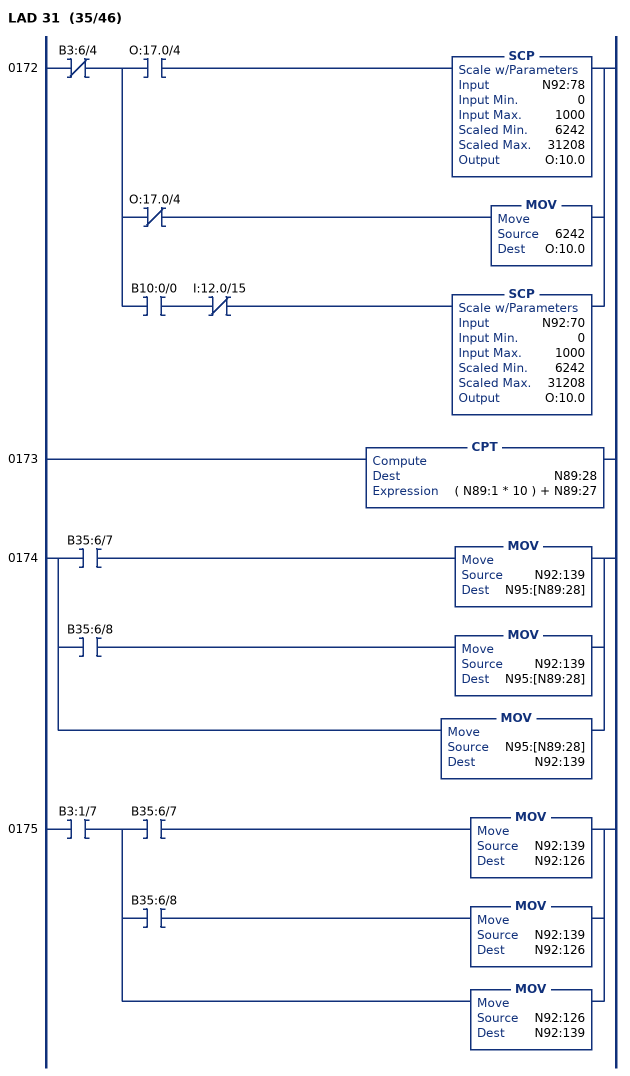
% Rung: 172 %
SOR XIO B3:6/4 BST XIC O:17.0/4 SCP N92:78 0 1000 6242 31208 O:10.0 NXB XIO O:17.0/4 MOV 6242 O:10.0 NXB XIC B10:0/0 XIO I:12.0/15 SCP N92:70 0 1000 6242 31208 O:10.0 BND EOR
% Rung: 173 %
SOR CPT N89:28 " ( N89:1 * 10 ) + N89:27 " EOR
% Rung: 174 %
SOR BST XIC B35:6/7 MOV N92:139 N95:[N89:28] NXB XIC B35:6/8 MOV N92:139 N95:[N89:28] NXB MOV N95:[N89:28] N92:139 BND EOR
% Rung: 175 %
SOR XIC B3:1/7 BST XIC B35:6/7 MOV N92:139 N92:126 NXB XIC B35:6/8 MOV N92:139 N92:126 NXB MOV N92:126 N92:139 BND EOR

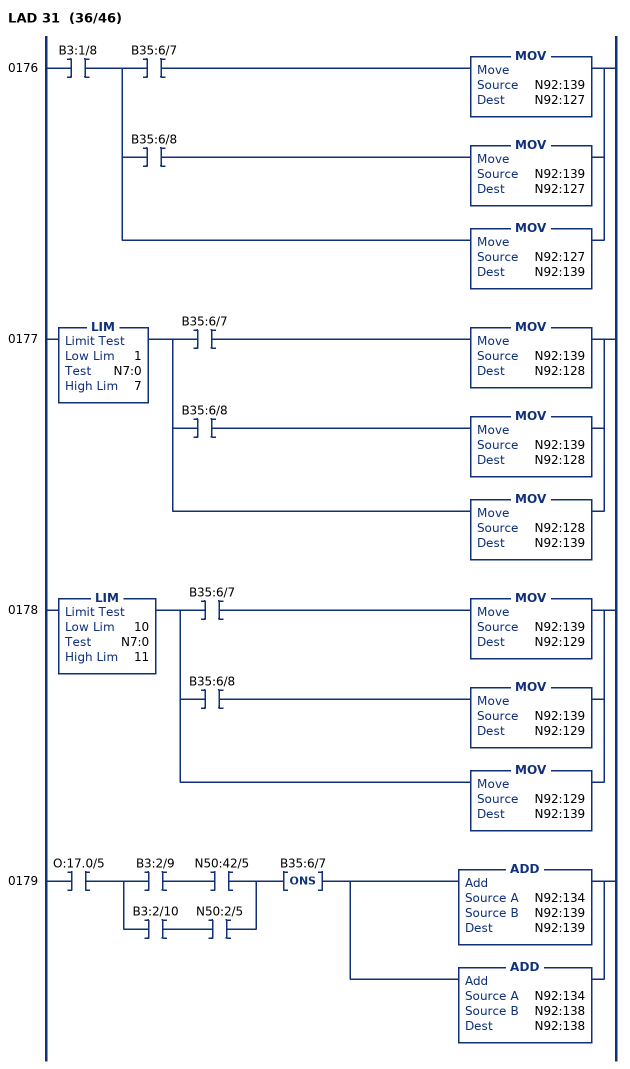
% Rung: 176 %
SOR XIC B3:1/8 BST XIC B35:6/7 MOV N92:139 N92:127 NXB XIC B35:6/8 MOV N92:139 N92:127 NXB MOV N92:127 N92:139 BND EOR
% Rung: 177 %
SOR LIM 1 N7:0 7 BST XIC B35:6/7 MOV N92:139 N92:128 NXB XIC B35:6/8 MOV N92:139 N92:128 NXB MOV N92:128 N92:139 BND EOR
% Rung: 178 %
SOR LIM 10 N7:0 11 BST XIC B35:6/7 MOV N92:139 N92:129 NXB XIC B35:6/8 MOV N92:139 N92:129 NXB MOV N92:129 N92:139 BND EOR
% Rung: 179 %
SOR XIC O:17.0/5 BST XIC B3:2/9 XIC N50:42/5 NXB XIC B3:2/10 XIC N50:2/5 BND OSR B35:6/7 BST ADD N92:134 N92:139 N92:139 NXB ADD N92:134 N92:138 N92:138 BND EOR

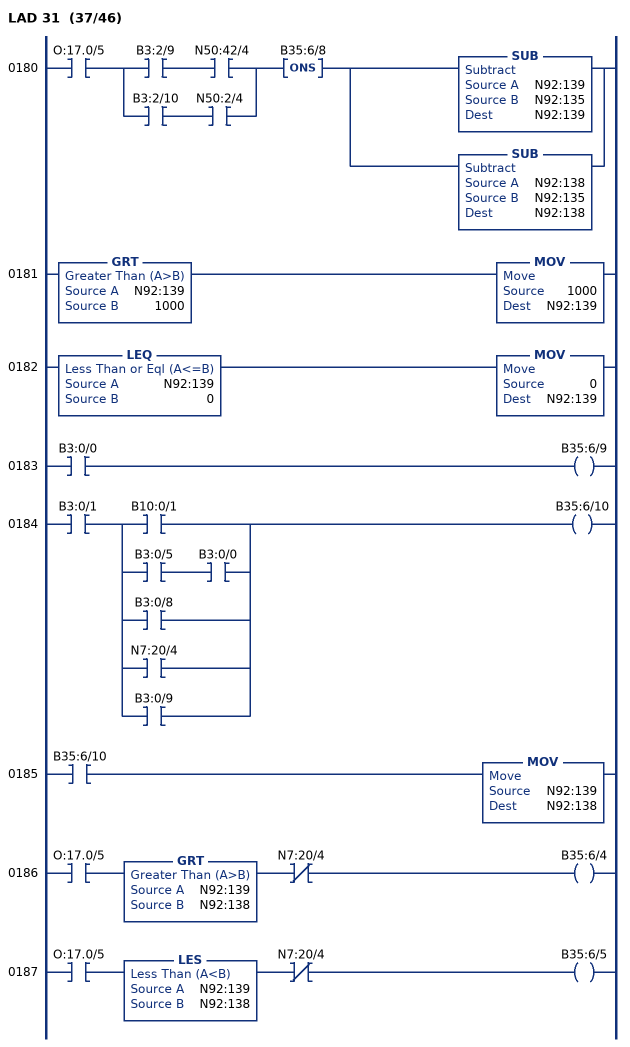
% Rung: 180 %
SOR XIC O:17.0/5 BST XIC B3:2/9 XIC N50:42/4 NXB XIC B3:2/10 XIC N50:2/4 BND OSR B35:6/8 BST SUB N92:139 N92:135 N92:139 NXB SUB N92:138 N92:135 N92:138 BND EOR
% Rung: 181 %
SOR GRT N92:139 1000 MOV 1000 N92:139 EOR
% Rung: 182 %
SOR LEQ N92:139 0 MOV 0 N92:139 EOR
% Rung: 183 %
SOR XIC B3:0/0 OTE B35:6/9 EOR
% Rung: 184 %
SOR XIC B3:0/1 BST XIC B10:0/1 NXB XIC B3:0/5 XIC B3:0/0 NXB XIC B3:0/8 NXB XIC N7:20/4 NXB XIC B3:0/9 BND OTE B35:6/10 EOR
% Rung: 185 %
SOR XIC B35:6/10 MOV N92:139 N92:138 EOR
% Rung: 186 %
SOR XIC O:17.0/5 GRT N92:139 N92:138 XIO N7:20/4 OTE B35:6/4 EOR
% Rung: 187 %
SOR XIC O:17.0/5 LES N92:139 N92:138 XIO N7:20/4 OTE B35:6/5 EOR

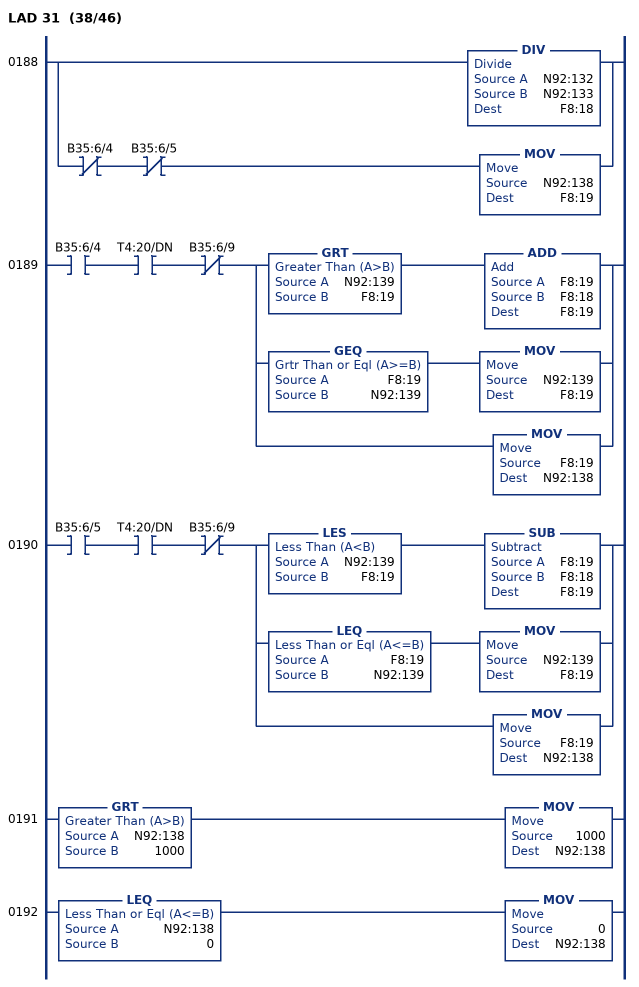
% Rung: 188 %
SOR BST DIV N92:132 N92:133 F8:18 NXB XIO B35:6/4 XIO B35:6/5 MOV N92:138 F8:19 BND EOR
% Rung: 189 %
SOR XIC B35:6/4 XIC T4:20/DN XIO B35:6/9 BST GRT N92:139 F8:19 ADD F8:19 F8:18 F8:19 NXB GEQ F8:19 N92:139 MOV N92:139 F8:19 NXB MOV F8:19 N92:138 BND EOR
% Rung: 190 %
SOR XIC B35:6/5 XIC T4:20/DN XIO B35:6/9 BST LES N92:139 F8:19 SUB F8:19 F8:18 F8:19 NXB LEQ F8:19 N92:139 MOV N92:139 F8:19 NXB MOV F8:19 N92:138 BND EOR
% Rung: 191 %
SOR GRT N92:138 1000 MOV 1000 N92:138 EOR
% Rung: 192 %
SOR LEQ N92:138 0 MOV 0 N92:138 EOR

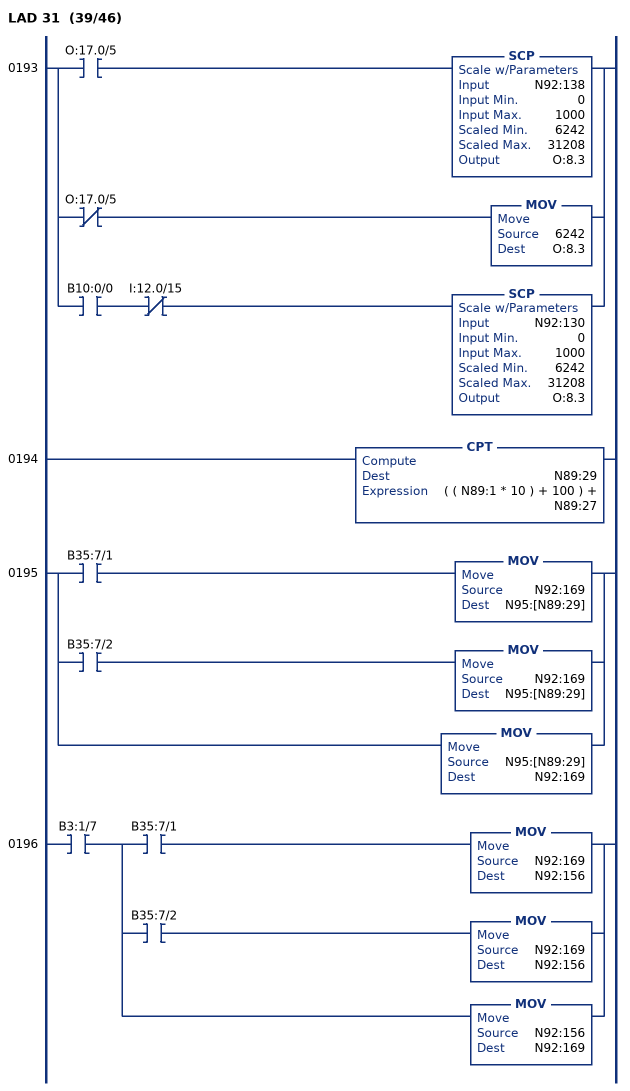
% Rung: 193 %
SOR BST XIC O:17.0/5 SCP N92:138 0 1000 6242 31208 O:8.3 NXB XIO O:17.0/5 MOV 6242 O:8.3 NXB XIC B10:0/0 XIO I:12.0/15 SCP N92:130 0 1000 6242 31208 O:8.3 BND EOR
% Rung: 194 %
SOR CPT N89:29 " ( ( N89:1 * 10 ) + 100 ) + N89:27 " EOR
% Rung: 195 %
SOR BST XIC B35:7/1 MOV N92:169 N95:[N89:29] NXB XIC B35:7/2 MOV N92:169 N95:[N89:29] NXB MOV N95:[N89:29] N92:169 BND EOR
% Rung: 196 %
SOR XIC B3:1/7 BST XIC B35:7/1 MOV N92:169 N92:156 NXB XIC B35:7/2 MOV N92:169 N92:156 NXB MOV N92:156 N92:169 BND EOR

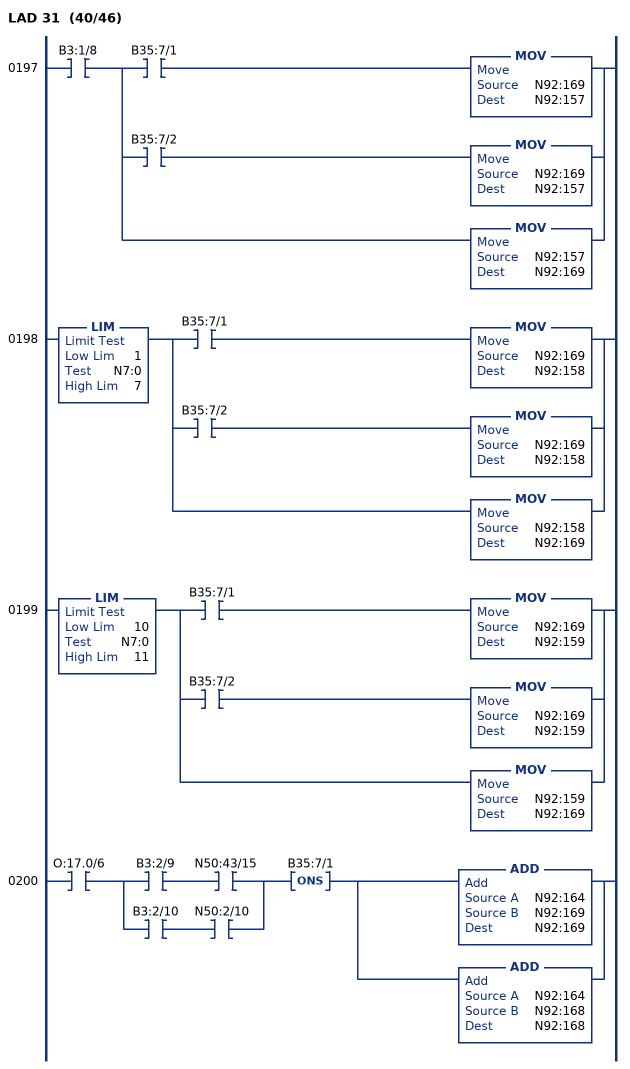
% Rung: 197 %
SOR XIC B3:1/8 BST XIC B35:7/1 MOV N92:169 N92:157 NXB XIC B35:7/2 MOV N92:169 N92:157 NXB MOV N92:157 N92:169 BND EOR
% Rung: 198 %
SOR LIM 1 N7:0 7 BST XIC B35:7/1 MOV N92:169 N92:158 NXB XIC B35:7/2 MOV N92:169 N92:158 NXB MOV N92:158 N92:169 BND EOR
% Rung: 199 %
SOR LIM 10 N7:0 11 BST XIC B35:7/1 MOV N92:169 N92:159 NXB XIC B35:7/2 MOV N92:169 N92:159 NXB MOV N92:159 N92:169 BND EOR
% Rung: 200 %
SOR XIC O:17.0/6 BST XIC B3:2/9 XIC N50:43/15 NXB XIC B3:2/10 XIC N50:2/10 BND OSR B35:7/1 BST ADD N92:164 N92:169 N92:169 NXB ADD N92:164 N92:168 N92:168 BND EOR

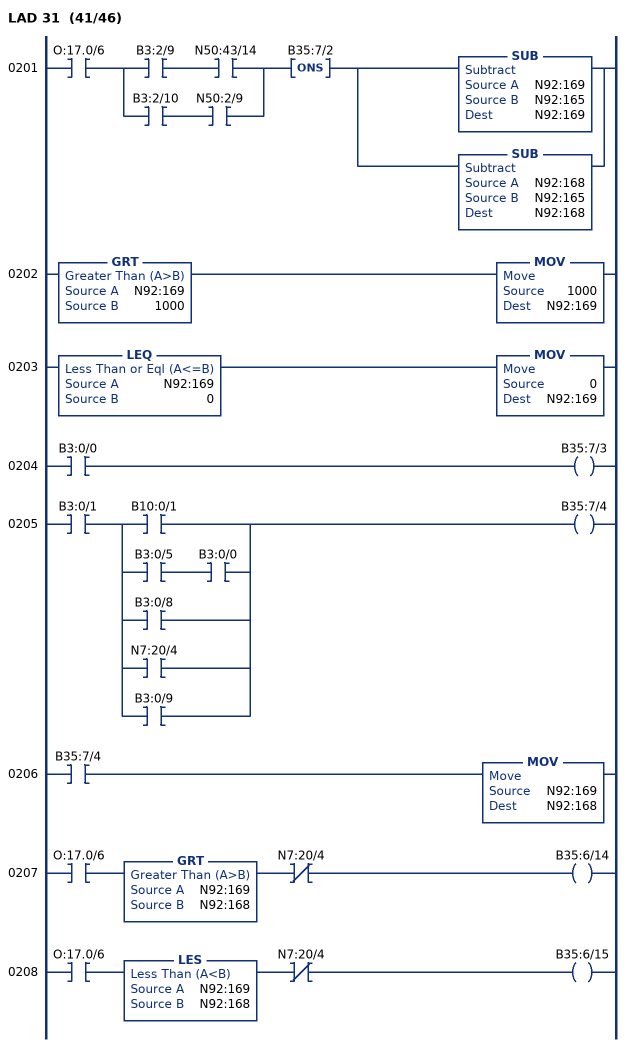
% Rung: 201 %
SOR XIC O:17.0/6 BST XIC B3:2/9 XIC N50:43/14 NXB XIC B3:2/10 XIC N50:2/9 BND OSR B35:7/2 BST SUB N92:169 N92:165 N92:169 NXB SUB N92:168 N92:165 N92:168 BND EOR
% Rung: 202 %
SOR GRT N92:169 1000 MOV 1000 N92:169 EOR
% Rung: 203 %
SOR LEQ N92:169 0 MOV 0 N92:169 EOR
% Rung: 204 %
SOR XIC B3:0/0 OTE B35:7/3 EOR
% Rung: 205 %
SOR XIC B3:0/1 BST XIC B10:0/1 NXB XIC B3:0/5 XIC B3:0/0 NXB XIC B3:0/8 NXB XIC N7:20/4 NXB XIC B3:0/9 BND OTE B35:7/4 EOR
% Rung: 206 %
SOR XIC B35:7/4 MOV N92:169 N92:168 EOR
% Rung: 207 %
SOR XIC O:17.0/6 GRT N92:169 N92:168 XIO N7:20/4 OTE B35:6/14 EOR
% Rung: 208 %
SOR XIC O:17.0/6 LES N92:169 N92:168 XIO N7:20/4 OTE B35:6/15 EOR

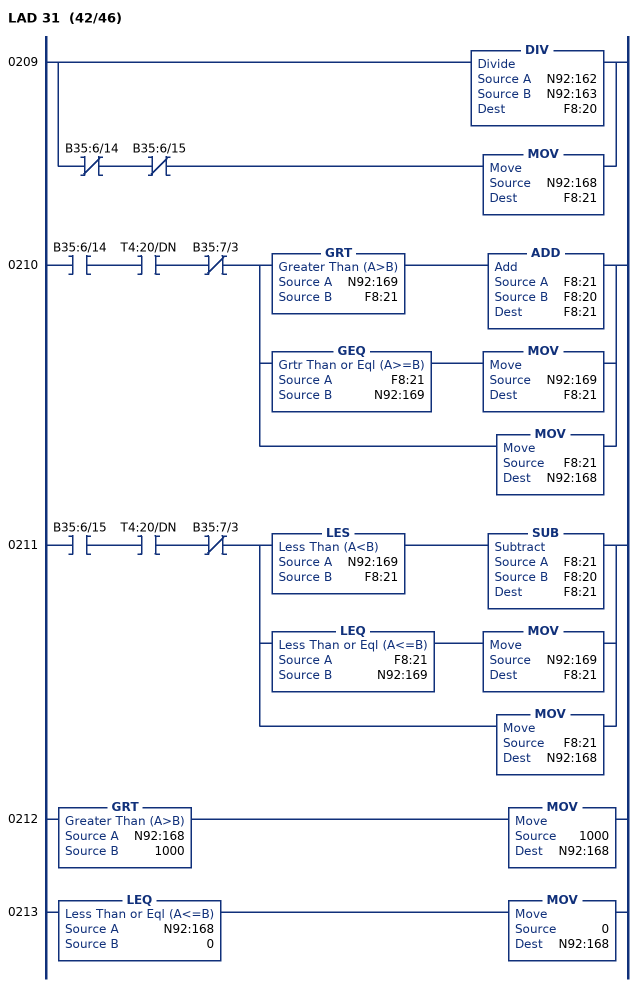
% Rung: 209 %
SOR BST DIV N92:162 N92:163 F8:20 NXB XIO B35:6/14 XIO B35:6/15 MOV N92:168 F8:21 BND EOR
% Rung: 210 %
SOR XIC B35:6/14 XIC T4:20/DN XIO B35:7/3 BST GRT N92:169 F8:21 ADD F8:21 F8:20 F8:21 NXB GEQ F8:21 N92:169 MOV N92:169 F8:21 NXB MOV F8:21 N92:168 BND EOR
% Rung: 211 %
SOR XIC B35:6/15 XIC T4:20/DN XIO B35:7/3 BST LES N92:169 F8:21 SUB F8:21 F8:20 F8:21 NXB LEQ F8:21 N92:169 MOV N92:169 F8:21 NXB MOV F8:21 N92:168 BND EOR
% Rung: 212 %
SOR GRT N92:168 1000 MOV 1000 N92:168 EOR
% Rung: 213 %
SOR LEQ N92:168 0 MOV 0 N92:168 EOR

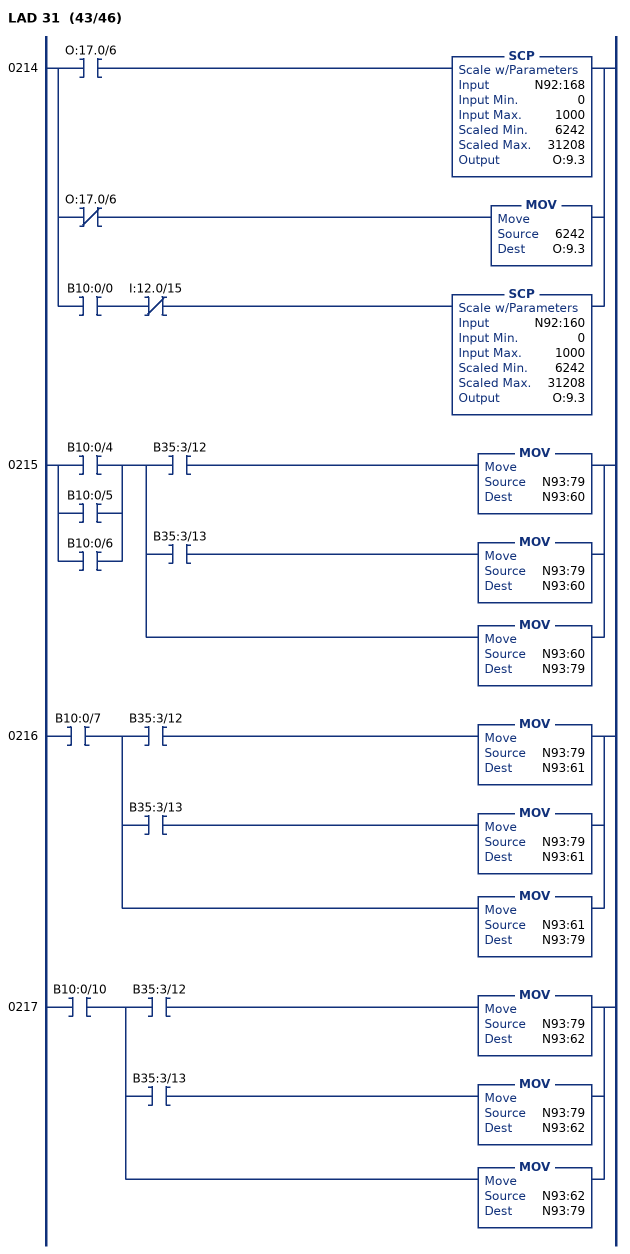
% Rung: 214 %
SOR BST XIC O:17.0/6 SCP N92:168 0 1000 6242 31208 O:9.3 NXB XIO O:17.0/6 MOV 6242 O:9.3 NXB XIC B10:0/0 XIO I:12.0/15 SCP N92:160 0 1000 6242 31208 O:9.3 BND EOR
% Rung: 215 %
SOR BST XIC B10:0/4 NXB XIC B10:0/5 NXB XIC B10:0/6 BND BST XIC B35:3/12 MOV N93:79 N93:60 NXB XIC B35:3/13 MOV N93:79 N93:60 NXB MOV N93:60 N93:79 BND EOR
% Rung: 216 %
SOR XIC B10:0/7 BST XIC B35:3/12 MOV N93:79 N93:61 NXB XIC B35:3/13 MOV N93:79 N93:61 NXB MOV N93:61 N93:79 BND EOR
% Rung: 217 %
SOR XIC B10:0/10 BST XIC B35:3/12 MOV N93:79 N93:62 NXB XIC B35:3/13 MOV N93:79 N93:62 NXB MOV N93:62 N93:79 BND EOR

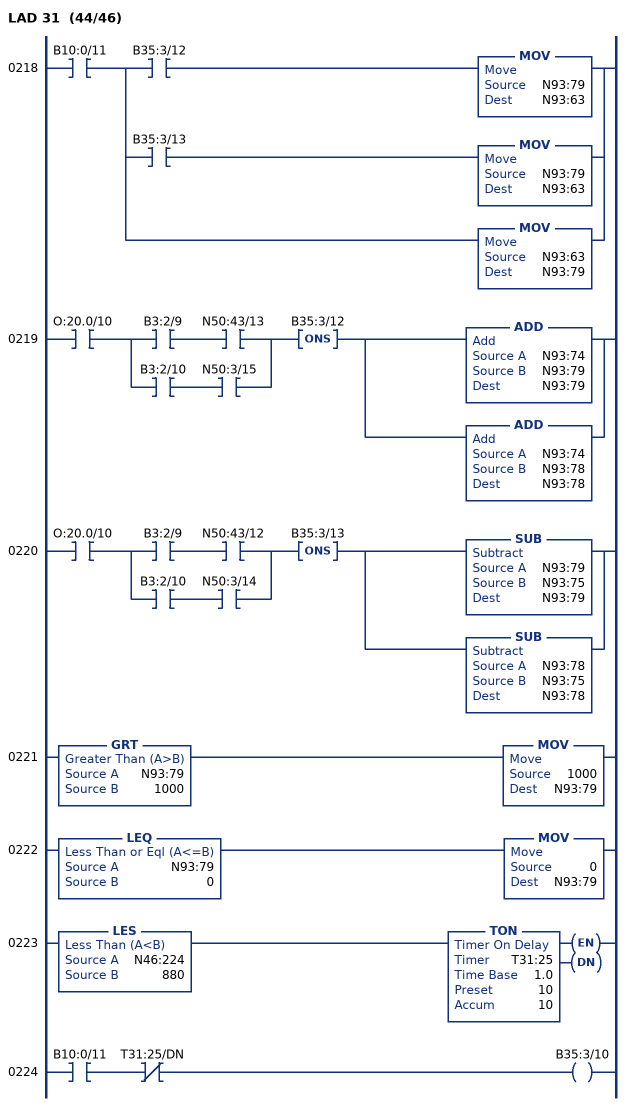
% Rung: 218 %
SOR XIC B10:0/11 BST XIC B35:3/12 MOV N93:79 N93:63 NXB XIC B35:3/13 MOV N93:79 N93:63 NXB MOV N93:63 N93:79 BND EOR
% Rung: 219 %
SOR XIC O:20.0/10 BST XIC B3:2/9 XIC N50:43/13 NXB XIC B3:2/10 XIC N50:3/15 BND OSR B35:3/12 BST ADD N93:74 N93:79 N93:79 NXB ADD N93:74 N93:78 N93:78 BND EOR
% Rung: 220 %
SOR XIC O:20.0/10 BST XIC B3:2/9 XIC N50:43/12 NXB XIC B3:2/10 XIC N50:3/14 BND OSR B35:3/13 BST SUB N93:79 N93:75 N93:79 NXB SUB N93:78 N93:75 N93:78 BND EOR
% Rung: 221 %
SOR GRT N93:79 1000 MOV 1000 N93:79 EOR
% Rung: 222 %
SOR LEQ N93:79 0 MOV 0 N93:79 EOR
% Rung: 223 %
SOR LES N46:224 880 TON T31:25 1.0 10 10 EOR
% Rung: 224 %
SOR XIC B10:0/11 XIO T31:25/DN OTE B35:3/10 EOR

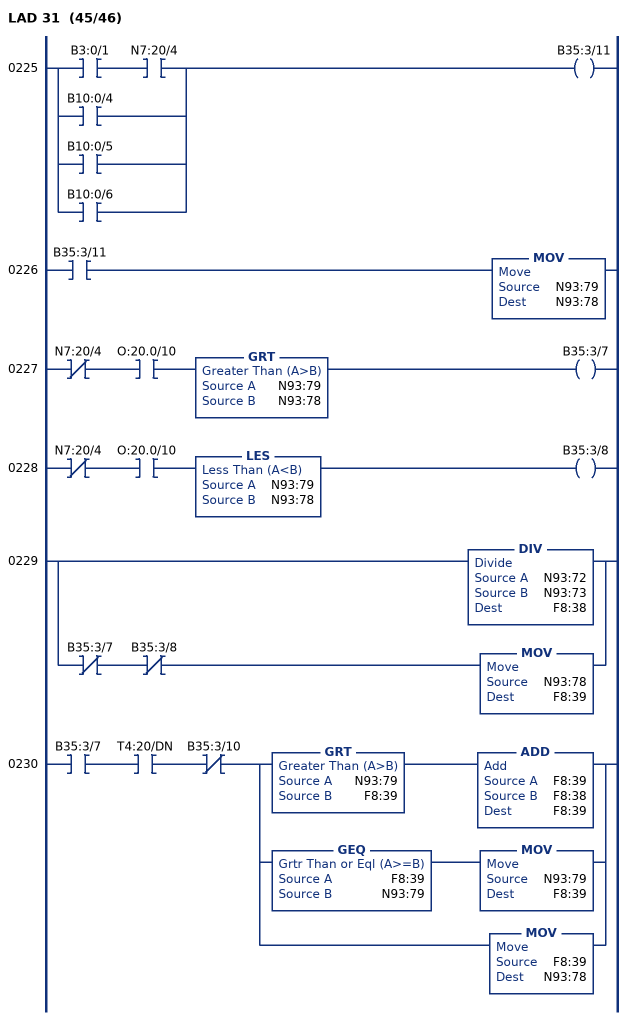
% Rung: 225 %
SOR BST XIC B3:0/1 XIC N7:20/4 NXB XIC B10:0/4 NXB XIC B10:0/5 NXB XIC B10:0/6 BND OTE B35:3/11 EOR
% Rung: 226 %
SOR XIC B35:3/11 MOV N93:79 N93:78 EOR
% Rung: 227 %
SOR XIO N7:20/4 XIC O:20.0/10 GRT N93:79 N93:78 OTE B35:3/7 EOR
% Rung: 228 %
SOR XIO N7:20/4 XIC O:20.0/10 LES N93:79 N93:78 OTE B35:3/8 EOR
% Rung: 229 %
SOR BST DIV N93:72 N93:73 F8:38 NXB XIO B35:3/7 XIO B35:3/8 MOV N93:78 F8:39 BND EOR
% Rung: 230 %
SOR XIC B35:3/7 XIC T4:20/DN XIO B35:3/10 BST GRT N93:79 F8:39 ADD F8:39 F8:38 F8:39 NXB GEQ F8:39 N93:79 MOV N93:79 F8:39 NXB MOV F8:39 N93:78 BND EOR

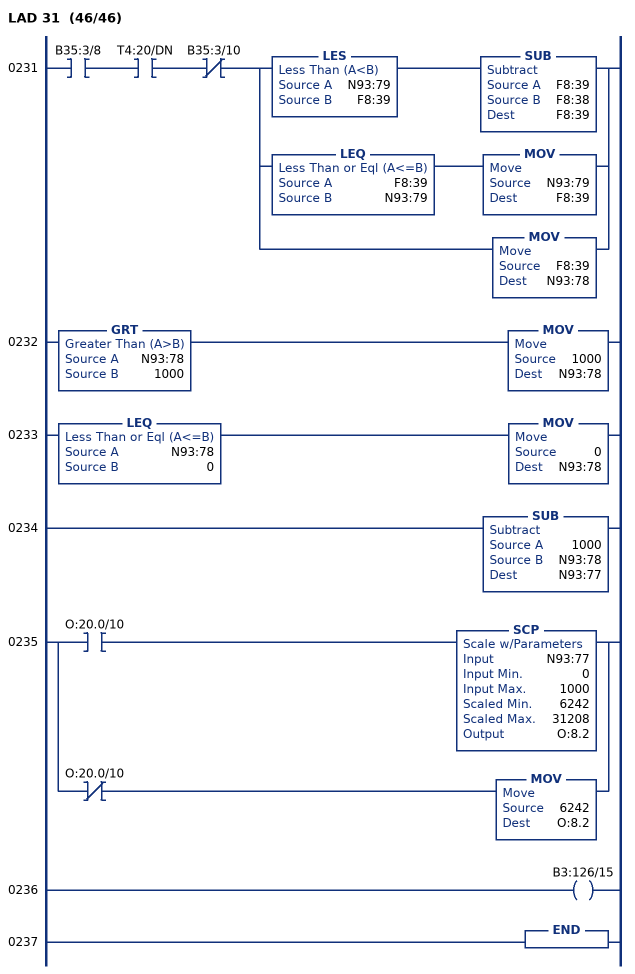
% Rung: 231 %
SOR XIC B35:3/8 XIC T4:20/DN XIO B35:3/10 BST LES N93:79 F8:39 SUB F8:39 F8:38 F8:39 NXB LEQ F8:39 N93:79 MOV N93:79 F8:39 NXB MOV F8:39 N93:78 BND EOR
% Rung: 232 %
SOR GRT N93:78 1000 MOV 1000 N93:78 EOR
% Rung: 233 %
SOR LEQ N93:78 0 MOV 0 N93:78 EOR
% Rung: 234 %
SOR SUB 1000 N93:78 N93:77 EOR
% Rung: 235 %
SOR BST XIC O:20.0/10 SCP N93:77 0 1000 6242 31208 O:8.2 NXB XIO O:20.0/10 MOV 6242 O:8.2 BND EOR
% Rung: 236 %
SOR OTE B3:126/15 EOR
% Rung: 237 %
SOR END EOR

LADDER 36
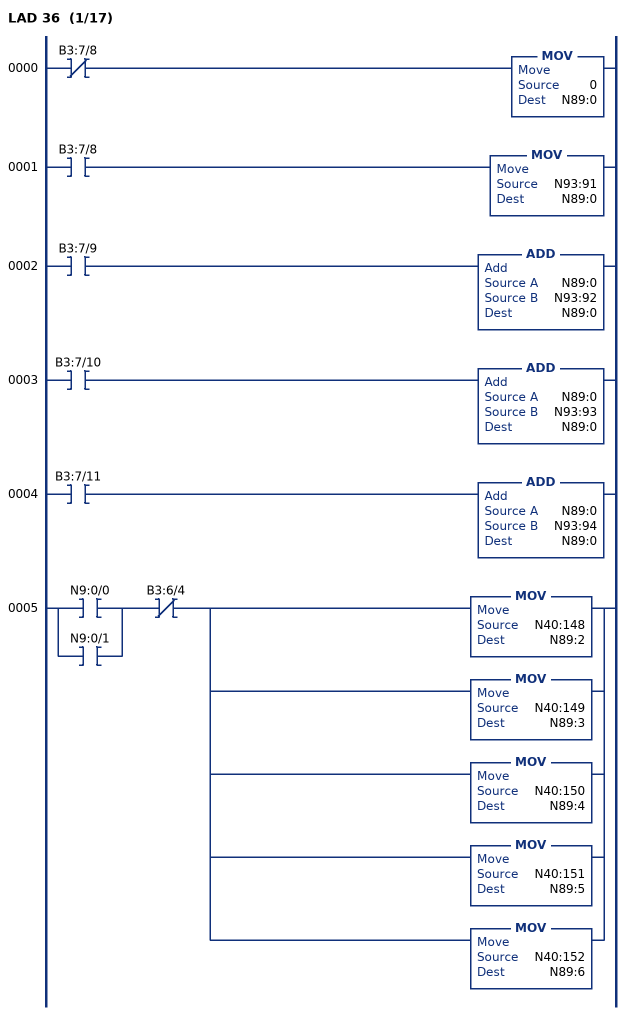
% Rung: 0 %
SOR XIO B3:7/8 MOV 0 N89:0 EOR
% Rung: 1 %
SOR XIC B3:7/8 MOV N93:91 N89:0 EOR
% Rung: 2 %
SOR XIC B3:7/9 ADD N89:0 N93:92 N89:0 EOR
% Rung: 3 %
SOR XIC B3:7/10 ADD N89:0 N93:93 N89:0 EOR
% Rung: 4 %
SOR XIC B3:7/11 ADD N89:0 N93:94 N89:0 EOR
% Rung: 5 %
SOR BST XIC N9:0/0 NXB XIC N9:0/1 BND XIO B3:6/4 BST MOV N40:148 N89:2 NXB MOV N40:149 N89:3 NXB MOV N40:150 N89:4 NXB MOV N40:151 N89:5 NXB MOV N40:152 N89:6 BND EOR

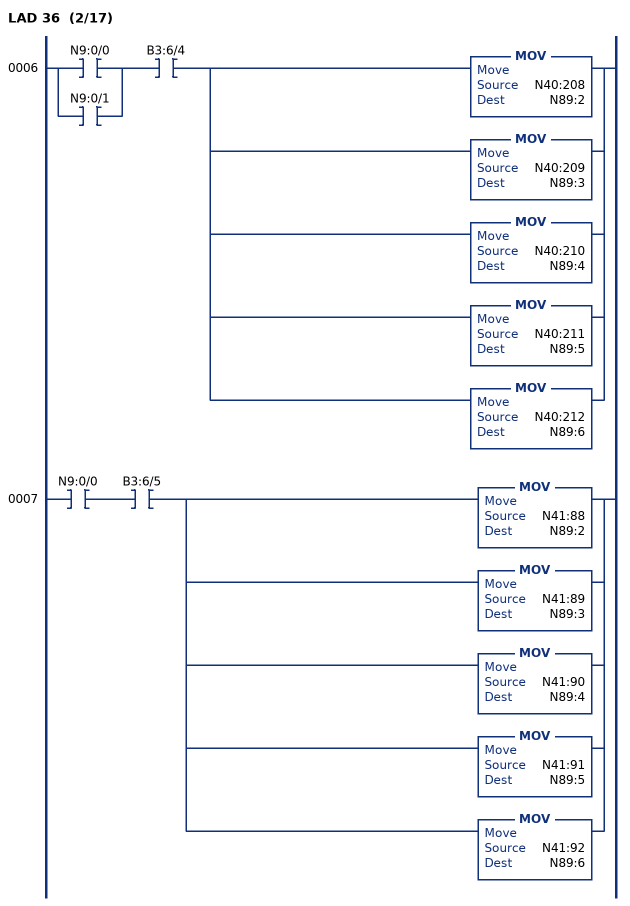
% Rung: 6 %
SOR BST XIC N9:0/0 NXB XIC N9:0/1 BND XIC B3:6/4 BST MOV N40:208 N89:2 NXB MOV N40:209 N89:3 NXB MOV N40:210 N89:4 NXB MOV N40:211 N89:5 NXB MOV N40:212 N89:6 BND EOR
% Rung: 7 %
SOR XIC N9:0/0 XIC B3:6/5 BST MOV N41:88 N89:2 NXB MOV N41:89 N89:3 NXB MOV N41:90 N89:4 NXB MOV N41:91 N89:5 NXB MOV N41:92 N89:6 BND EOR

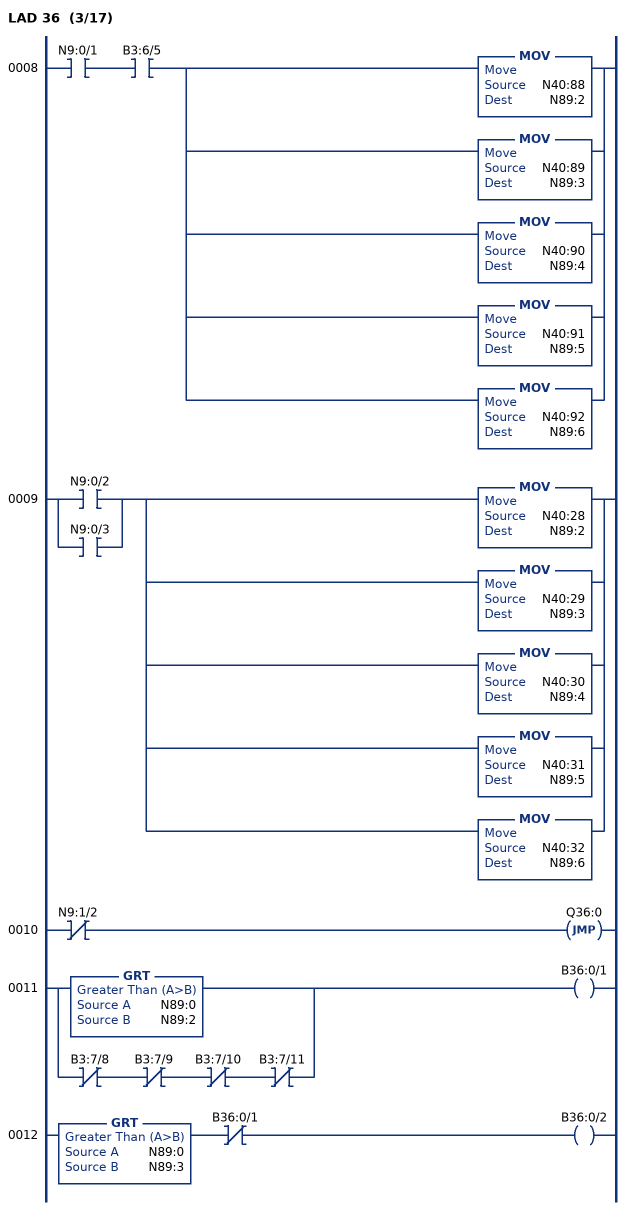
% Rung: 8 %
SOR XIC N9:0/1 XIC B3:6/5 BST MOV N40:88 N89:2 NXB MOV N40:89 N89:3 NXB MOV N40:90 N89:4 NXB MOV N40:91 N89:5 NXB MOV N40:92 N89:6 BND EOR
% Rung: 9 %
SOR BST XIC N9:0/2 NXB XIC N9:0/3 BND BST MOV N40:28 N89:2 NXB MOV N40:29 N89:3 NXB MOV N40:30 N89:4 NXB MOV N40:31 N89:5 NXB MOV N40:32 N89:6 BND EOR
% Rung: 10 %
SOR XIO N9:1/2 JMP Q36:0 EOR
% Rung: 11 %
SOR BST GRT N89:0 N89:2 NXB XIO B3:7/8 XIO B3:7/9 XIO B3:7/10 XIO B3:7/11 BND OTE B36:0/1 EOR
% Rung: 12 %
SOR GRT N89:0 N89:3 XIO B36:0/1 OTE B36:0/2 EOR

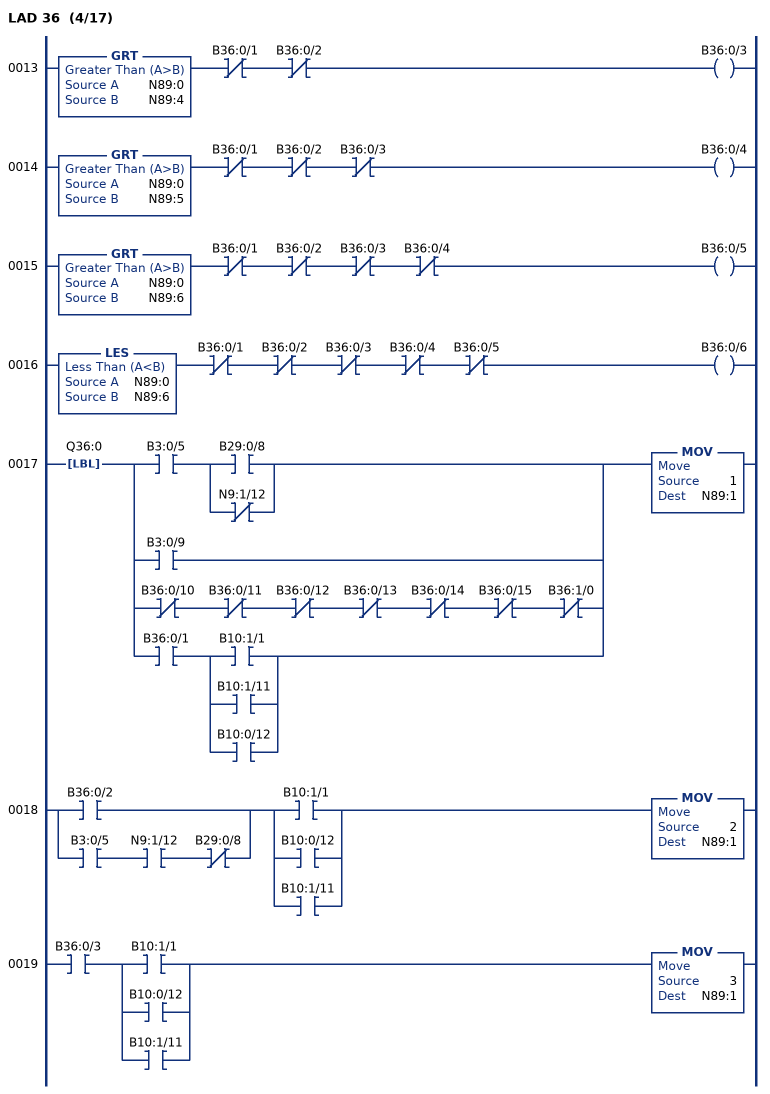
% Rung: 13 %
SOR GRT N89:0 N89:4 XIO B36:0/1 XIO B36:0/2 OTE B36:0/3 EOR
% Rung: 14 %
SOR GRT N89:0 N89:5 XIO B36:0/1 XIO B36:0/2 XIO B36:0/3 OTE B36:0/4 EOR
% Rung: 15 %
SOR GRT N89:0 N89:6 XIO B36:0/1 XIO B36:0/2 XIO B36:0/3 XIO B36:0/4 OTE B36:0/5 EOR
% Rung: 16 %
SOR LES N89:0 N89:6 XIO B36:0/1 XIO B36:0/2 XIO B36:0/3 XIO B36:0/4 XIO B36:0/5 OTE B36:0/6 EOR
% Rung: 17 %
SOR LBL Q36:0 BST XIC B3:0/5 BST XIC B29:0/8 NXB XIO N9:1/12 BND NXB XIC B3:0/9 NXB XIO B36:0/10 XIO B36:0/11 XIO B36:0/12 XIO B36:0/13 XIO B36:0/14 XIO B36:0/15 XIO B36:1/0 NXB XIC B36:0/1 BST XIC B10:1/1 NXB XIC B10:1/11 NXB XIC B10:0/12 BND BND MOV 1 N89:1 EOR
% Rung: 18 %
SOR BST XIC B36:0/2 NXB XIC B3:0/5 XIC N9:1/12 XIO B29:0/8 BND BST XIC B10:1/1 NXB XIC B10:0/12 NXB XIC B10:1/11 BND MOV 2 N89:1 EOR
% Rung: 19 %
SOR XIC B36:0/3 BST XIC B10:1/1 NXB XIC B10:0/12 NXB XIC B10:1/11 BND MOV 3 N89:1 EOR

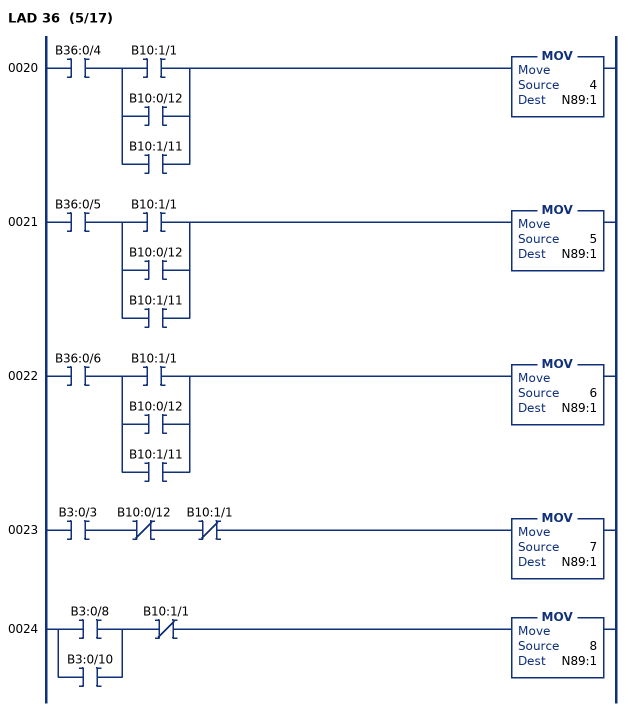
% Rung: 20 %
SOR XIC B36:0/4 BST XIC B10:1/1 NXB XIC B10:0/12 NXB XIC B10:1/11 BND MOV 4 N89:1 EOR
% Rung: 21 %
SOR XIC B36:0/5 BST XIC B10:1/1 NXB XIC B10:0/12 NXB XIC B10:1/11 BND MOV 5 N89:1 EOR
% Rung: 22 %
SOR XIC B36:0/6 BST XIC B10:1/1 NXB XIC B10:0/12 NXB XIC B10:1/11 BND MOV 6 N89:1 EOR
% Rung: 23 %
SOR XIC B3:0/3 XIO B10:0/12 XIO B10:1/1 MOV 7 N89:1 EOR
% Rung: 24 %
SOR BST XIC B3:0/8 NXB XIC B3:0/10 BND XIO B10:1/1 MOV 8 N89:1 EOR

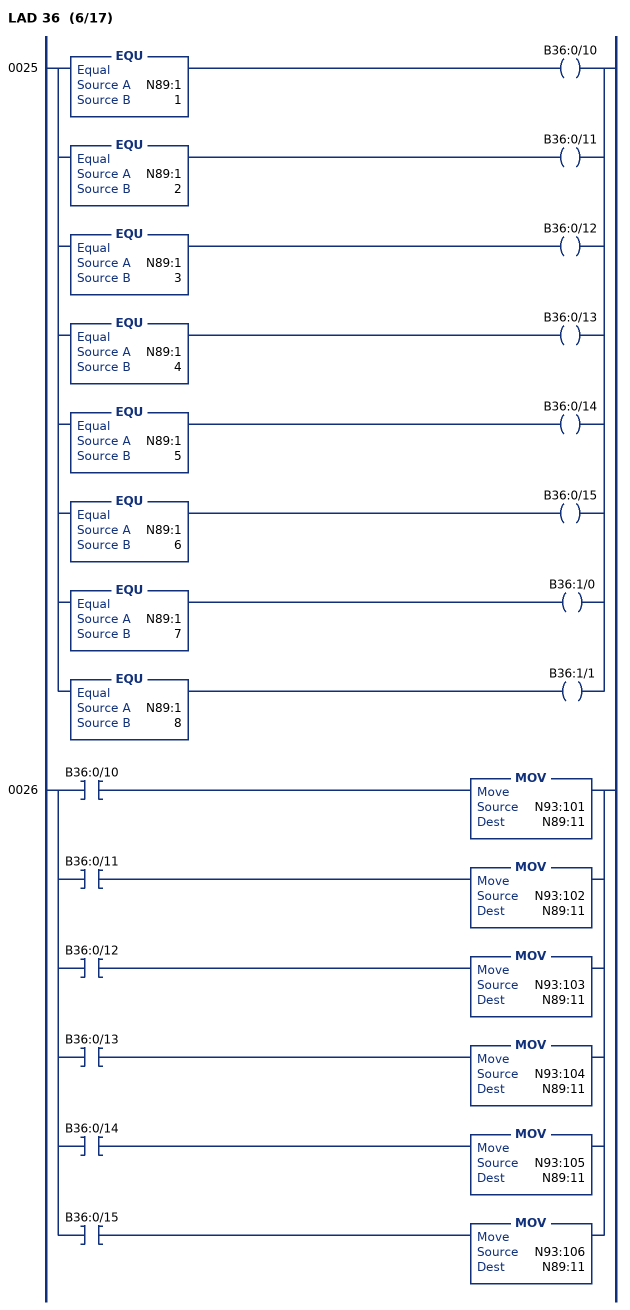
% Rung: 25 %
SOR BST EQU N89:1 1 OTE B36:0/10 NXB EQU N89:1 2 OTE B36:0/11 NXB EQU N89:1 3 OTE B36:0/12 NXB EQU N89:1 4 OTE B36:0/13 NXB EQU N89:1 5 OTE B36:0/14 NXB EQU N89:1 6 OTE B36:0/15 NXB EQU N89:1 7 OTE B36:1/0 NXB EQU N89:1 8 OTE B36:1/1 BND EOR
% Rung: 26 %
SOR BST XIC B36:0/10 MOV N93:101 N89:11 NXB XIC B36:0/11 MOV N93:102 N89:11 NXB XIC B36:0/12 MOV N93:103 N89:11 NXB XIC B36:0/13 MOV N93:104 N89:11 NXB XIC B36:0/14 MOV N93:105 N89:11 NXB XIC B36:0/15 MOV N93:106 N89:11 BND EOR

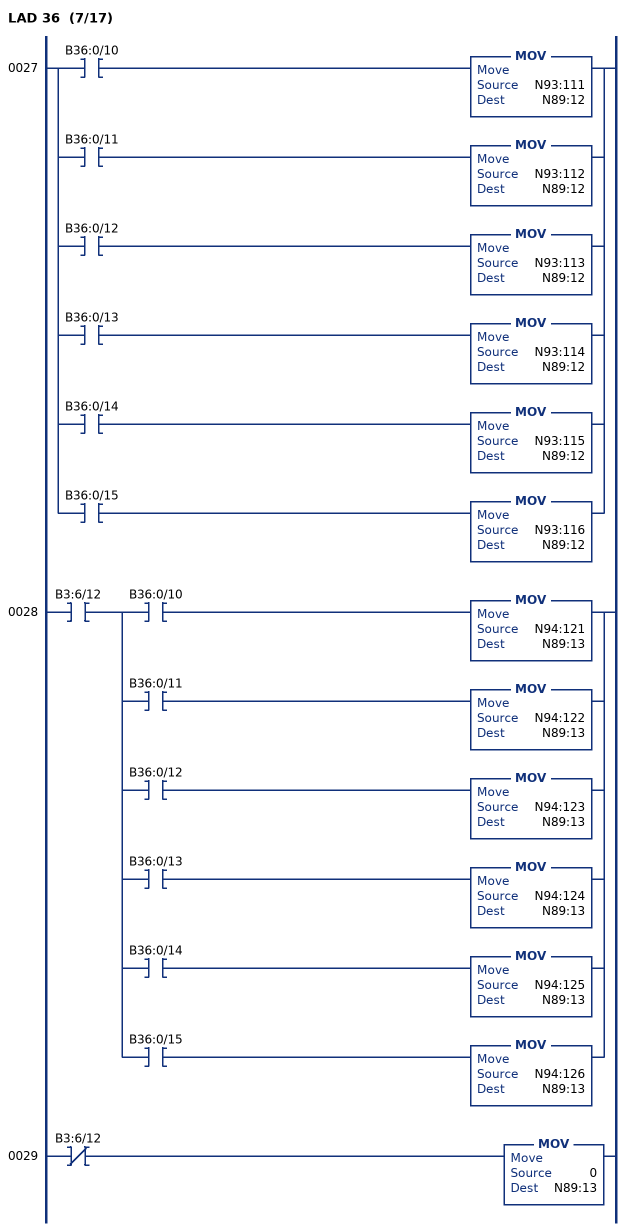
% Rung: 27 %
SOR BST XIC B36:0/10 MOV N93:111 N89:12 NXB XIC B36:0/11 MOV N93:112 N89:12 NXB XIC B36:0/12 MOV N93:113 N89:12 NXB XIC B36:0/13 MOV N93:114 N89:12 NXB XIC B36:0/14 MOV N93:115 N89:12 NXB XIC B36:0/15 MOV N93:116 N89:12 BND EOR
% Rung: 28 %
SOR XIC B3:6/12 BST XIC B36:0/10 MOV N94:121 N89:13 NXB XIC B36:0/11 MOV N94:122 N89:13 NXB XIC B36:0/12 MOV N94:123 N89:13 NXB XIC B36:0/13 MOV N94:124 N89:13 NXB XIC B36:0/14 MOV N94:125 N89:13 NXB XIC B36:0/15 MOV N94:126 N89:13 BND EOR
% Rung: 29 %
SOR XIO B3:6/12 MOV 0 N89:13 EOR

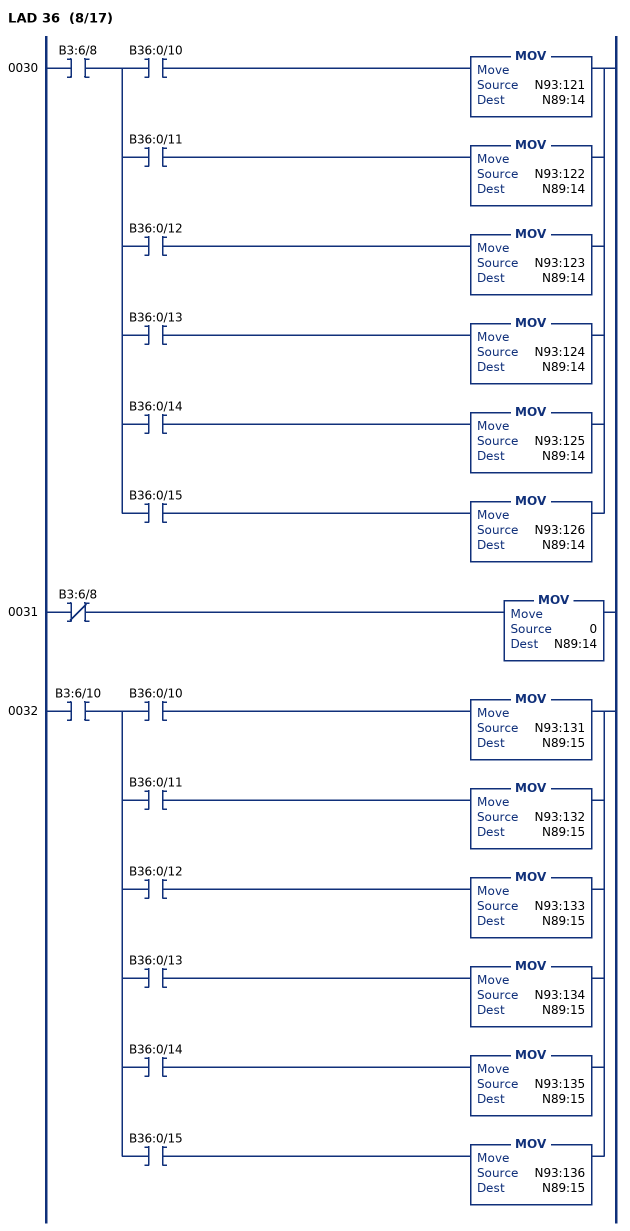
% Rung: 30 %
SOR XIC B3:6/8 BST XIC B36:0/10 MOV N93:121 N89:14 NXB XIC B36:0/11 MOV N93:122 N89:14 NXB XIC B36:0/12 MOV N93:123 N89:14 NXB XIC B36:0/13 MOV N93:124 N89:14 NXB XIC B36:0/14 MOV N93:125 N89:14 NXB XIC B36:0/15 MOV N93:126 N89:14 BND EOR
% Rung: 31 %
SOR XIO B3:6/8 MOV 0 N89:14 EOR
% Rung: 32 %
SOR XIC B3:6/10 BST XIC B36:0/10 MOV N93:131 N89:15 NXB XIC B36:0/11 MOV N93:132 N89:15 NXB XIC B36:0/12 MOV N93:133 N89:15 NXB XIC B36:0/13 MOV N93:134 N89:15 NXB XIC B36:0/14 MOV N93:135 N89:15 NXB XIC B36:0/15 MOV N93:136 N89:15 BND EOR

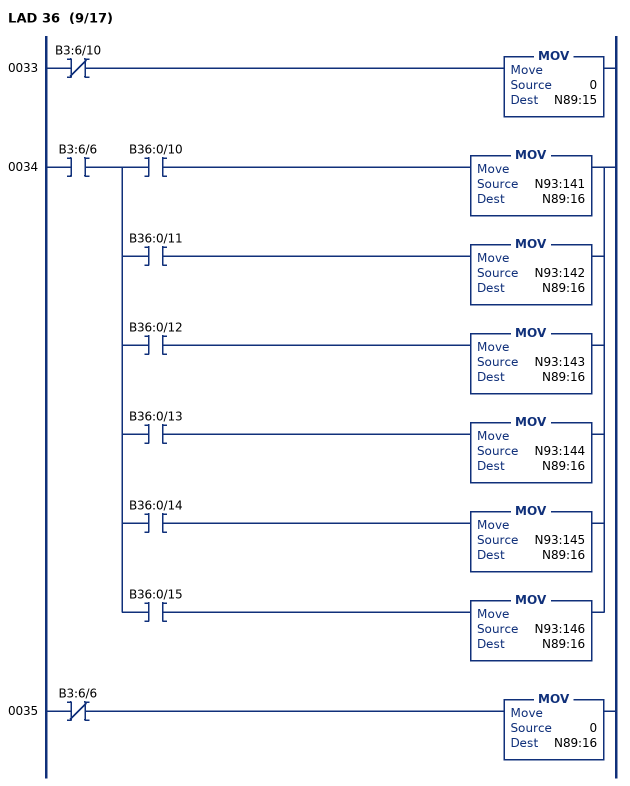
% Rung: 33 %
SOR XIO B3:6/10 MOV 0 N89:15 EOR
% Rung: 34 %
SOR XIC B3:6/6 BST XIC B36:0/10 MOV N93:141 N89:16 NXB XIC B36:0/11 MOV N93:142 N89:16 NXB XIC B36:0/12 MOV N93:143 N89:16 NXB XIC B36:0/13 MOV N93:144 N89:16 NXB XIC B36:0/14 MOV N93:145 N89:16 NXB XIC B36:0/15 MOV N93:146 N89:16 BND EOR
% Rung: 35 %
SOR XIO B3:6/6 MOV 0 N89:16 EOR

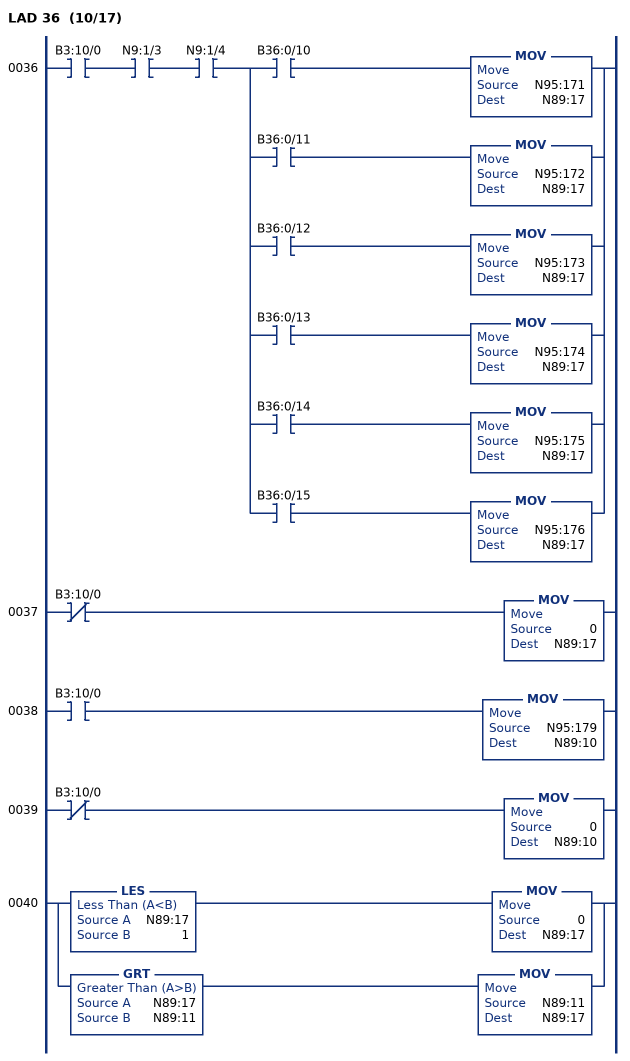
% Rung: 36 %
SOR XIC B3:10/0 XIC N9:1/3 XIC N9:1/4 BST XIC B36:0/10 MOV N95:171 N89:17 NXB XIC B36:0/11 MOV N95:172 N89:17 NXB XIC B36:0/12 MOV N95:173 N89:17 NXB XIC B36:0/13 MOV N95:174 N89:17 NXB XIC B36:0/14 MOV N95:175 N89:17 NXB XIC B36:0/15 MOV N95:176 N89:17 BND EOR
% Rung: 37 %
SOR XIO B3:10/0 MOV 0 N89:17 EOR
% Rung: 38 %
SOR XIC B3:10/0 MOV N95:179 N89:10 EOR
% Rung: 39 %
SOR XIO B3:10/0 MOV 0 N89:10 EOR
% Rung: 40 %
SOR BST LES N89:17 1 MOV 0 N89:17 NXB GRT N89:17 N89:11 MOV N89:11 N89:17 BND EOR

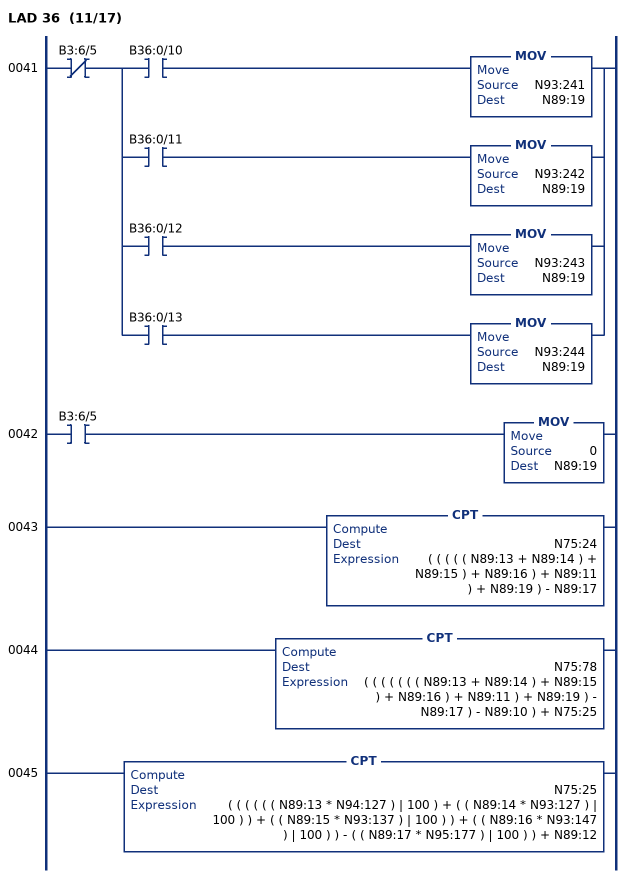
% Rung: 41 %
SOR XIO B3:6/5 BST XIC B36:0/10 MOV N93:241 N89:19 NXB XIC B36:0/11 MOV N93:242 N89:19 NXB XIC B36:0/12 MOV N93:243 N89:19 NXB XIC B36:0/13 MOV N93:244 N89:19 BND EOR
% Rung: 42 %
SOR XIC B3:6/5 MOV 0 N89:19 EOR
% Rung: 43 %
SOR CPT N75:24 " ( ( ( ( ( N89:13 + N89:14 ) + N89:15 ) + N89:16 ) + N89:11 ) + N89:19 ) - N89:17 " EOR
% Rung: 44 %
SOR CPT N75:78 " ( ( ( ( ( ( ( N89:13 + N89:14 ) + N89:15 ) + N89:16 ) + N89:11 ) + N89:19 ) - N89:17 ) - N89:10 ) + N75:25 " EOR
% Rung: 45 %
SOR CPT N75:25 " ( ( ( ( ( ( N89:13 * N94:127 ) | 100 ) + ( ( N89:14 * N93:127 ) | 100 ) ) + ( ( N89:15 * N93:137 ) | 100 ) ) + ( ( N89:16 * N93:147 ) | 100 ) ) - ( ( N89:17 * N95:177 ) | 100 ) ) + N89:12 " EOR

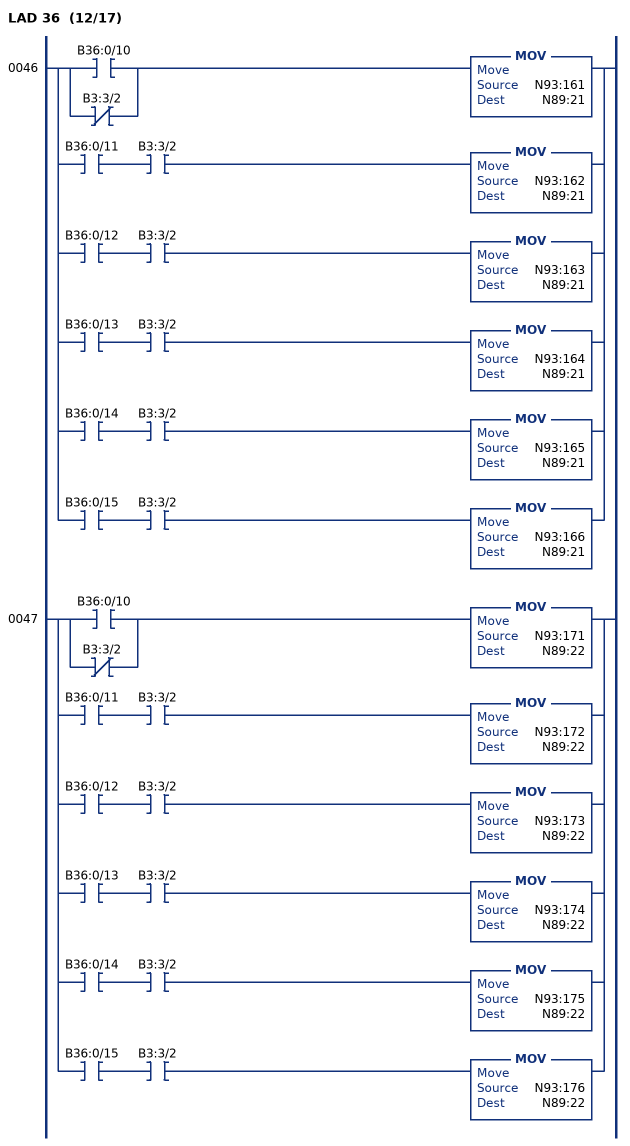
% Rung: 46 %
SOR BST BST XIC B36:0/10 NXB XIO B3:3/2 BND MOV N93:161 N89:21 NXB XIC B36:0/11 XIC B3:3/2 MOV N93:162 N89:21 NXB XIC B36:0/12 XIC B3:3/2 MOV N93:163 N89:21 NXB XIC B36:0/13 XIC B3:3/2 MOV N93:164 N89:21 NXB XIC B36:0/14 XIC B3:3/2 MOV N93:165 N89:21 NXB XIC B36:0/15 XIC B3:3/2 MOV N93:166 N89:21 BND EOR
% Rung: 47 %
SOR BST BST XIC B36:0/10 NXB XIO B3:3/2 BND MOV N93:171 N89:22 NXB XIC B36:0/11 XIC B3:3/2 MOV N93:172 N89:22 NXB XIC B36:0/12 XIC B3:3/2 MOV N93:173 N89:22 NXB XIC B36:0/13 XIC B3:3/2 MOV N93:174 N89:22 NXB XIC B36:0/14 XIC B3:3/2 MOV N93:175 N89:22 NXB XIC B36:0/15 XIC B3:3/2 MOV N93:176 N89:22 BND EOR

